{attribute 'qualified_only'}
{attribute 'strict'}
{attribute 'to_string'}
TYPE OPC_UA_COMMUNICATOR_STATE :
(
	IDLE,
	CONNECT,
	GET_NAMESPACE_INDEX,
	GET_NODE_HANDLE,
	PERFORM_ACTION,
	WAIT_FOR_NEXT_CYCLE,
	RELEASE_NODE_HANDLE,
	DISCONNECT
);
END_TYPE

(* stored: Version 1.1.0.1
   DUT OPC_UA_COMMUNICATOR_STATE: Id {90deca77-22a1-4000-b9fc-44c1c9e1d6c5} *)
